Fanuc KAREL source: VAR_LIST.kl

PROGRAM T
%NOLOCKGROUP
VAR
 v0 : STRING[40]
 v1 : STRING[40]
 v2 : INTEGER
 v3 : INTEGER
 v4 : INTEGER
 v5 : ARRAY[10] OF STRING[40]
 v6 : INTEGER
 v7 : INTEGER
BEGIN
 VAR_LIST(v0, v1, v2, v3, v4, v5, v6, v7)
END T
